FUNCTION_BLOCK FB_DriveReverse EXTENDS FB_Drive IMPLEMENTS I_DriveReverse

VAR
	_contactorReverse		: ContactorReverse;	// załącz/wyłącz stycznik do tyłu silnika

END_VAR

//SUPER^();

METHOD StatusState : STRING
VAR_INPUT
END_VAR
// ustaw stan zmiennej LED Taurusa w TANGO SCADA (zmiana koloru diody predefiniowana tekstem) oraz label statusu jako tekst
// zliczaj czas pracy gdy napęd jest uruchomiony


IF _termFuse.IsActive THEN
		_supplyLed.State := TRUE;
		_stateLabel.Text := 'ON';
		_statusLabel.Text := 'Napęd jest w gotowości';	

	IF _contactor.State THEN
		_stateLabel.Text := 'RUNNING';
		_statusLabel.Text := 'Napęd jest uruchomiony do przodu';
		
		// start count work time
		WorkTimelabel();
	END_IF
	
	IF _contactorReverse.State THEN
		_stateLabel.Text := 'RUNNING';
		_statusLabel.Text := 'Napęd jest uruchomiony do tyłu';
		
		// start count work time
		WorkTimelabel();
	END_IF
	
	

ELSE
		_supplyLed.State := FALSE;
		_stateLabel.Text := 'OFF';
		_statusLabel.Text := 'Napęd jest wyłączony';

	IF _contactor.State OR _contactorReverse.State THEN
		_stateLabel.Text := 'FAULT';
		_statusLabel.Text := 'Zadziałał wyłacznik silnikowy';
	END_IF

END_IF
END_METHOD

METHOD SwitchReverseOff : BOOL
_contactorReverse.State := False;
END_METHOD

METHOD SwitchReverseOn : BOOL
_contactorReverse.State := TRUE;
END_METHOD

END_FUNCTION_BLOCK

(* stored: Version 1.1.0.1, ProductVersion 3.1.4024.12
   POU FB_DriveReverse: Id {e7f5413c-681f-401c-af50-970535df7710}, SpecialFunc None
   Method StatusState: Id {9134f4c8-a297-452b-a6ad-a83f0aad6a9c}
   Method SwitchReverseOff: Id {1bf8401f-e92a-45bf-8d9b-1f25e75c2802}
   Method SwitchReverseOn: Id {d0c55b9b-ce07-4e2d-8242-0831ea7d7140} *)
